{attribute 'qualified_only'}
VAR_GLOBAL
END_VAR

(* stored: Version 1.1.0.1, ProductVersion 3.1.4022.18
   GVL GVL: Id {b4d3eb96-00fb-43dd-b0eb-e06a044b2e61} *)
